FUNCTION_BLOCK E_CTUD
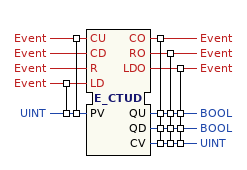
  EVENT_INPUT
    CU WITH PV;
    CD;
    R;
    LD WITH PV;
  END_EVENT
  EVENT_OUTPUT
    CO WITH QU, CV, QD;
    RO WITH QU, CV, QD;
    LDO WITH QU, QD, CV;
  END_EVENT
  VAR_INPUT
    PV : UINT;
  END_VAR
  VAR_OUTPUT
    QU : BOOL;
    QD : BOOL;
    CV : UINT;
  END_VAR
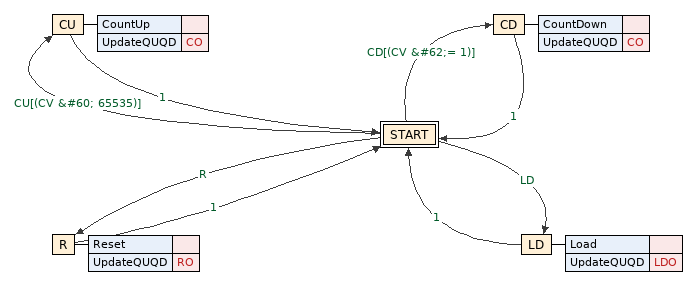
  EC_STATES
    START;
    CU : CountUp, UpdateQUQD -> CO;
    R : Reset, UpdateQUQD -> RO;
    CD : CountDown, UpdateQUQD -> CO;
    LD : Load, UpdateQUQD -> LDO;
  END_STATES
  EC_TRANSITIONS
    START TO CU := CU[(CV &#60; 65535)];
    CU TO START := 1;
    START TO R := R;
    R TO START := 1;
    START TO CD := CD[(CV &#62;= 1)];
    CD TO START := 1;
    START TO LD := LD;
    LD TO START := 1;
  END_TRANSITIONS
  ALGORITHM CountUp IN ST:
CV := CV + 1;&#38;#10;
  END_ALGORITHM
  ALGORITHM Reset IN ST:
CV := 0;&#38;#10;
  END_ALGORITHM
  ALGORITHM Load IN ST:
CV := PV;&#38;#10;
  END_ALGORITHM
  ALGORITHM UpdateQUQD IN ST:
QU := (CV &#62;= PV);&#38;#10;QD := (CV &#60;= 0);&#38;#10;
  END_ALGORITHM
  ALGORITHM CountDown IN ST:
CV := CV - 1;&#38;#10;
  END_ALGORITHM
END_FUNCTION_BLOCK
